ABB RAPID module: GM2694_96_A.mod

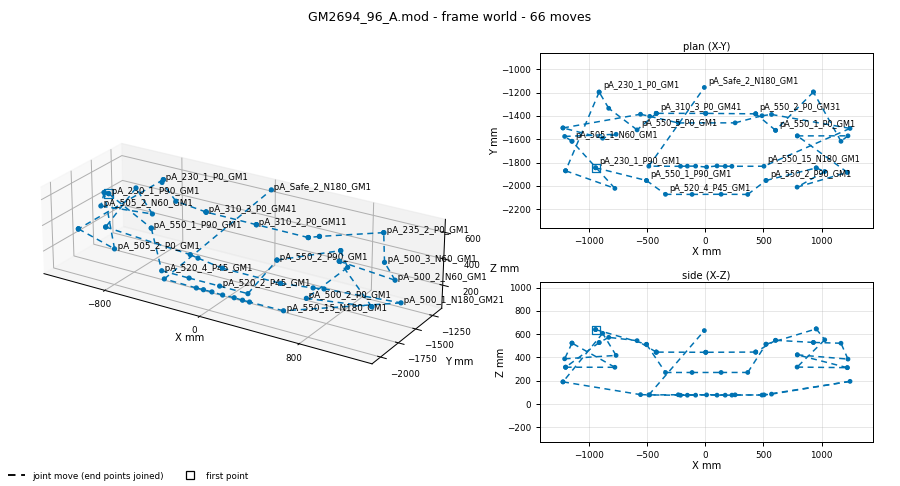
[picture p0: tool path of GM2694_96_A.mod in frame world, 66 of 72 moves have a stored position in this frame; points joined in program order, loops and branches not executed]
MODULE GM2694_96_A
	!Tool number
	TASK PERS wobjdata wobj_A_FD2:=[FALSE,TRUE,"STN2",[[0,0,0],[1,0,0,0]],[[-1.05287,-1136.44,433.383],[0.00113552,3.506E-06,-8.93971E-05,0.999999]]];

	!bailing room Jan 2013 Pad points
	CONST robtarget pTool_A_X1_FD2:=[[802.99,-1138.28,433.37],[1,2.43485E-05,-1.64211E-05,1.10567E-05],[-1,0,-1,1],[9E+09,9E+09,9E+09,9E+09,0.0243479,9E+09]];
	CONST robtarget pTool_A_X2_FD2:=[[-803.79,-1134.62,433.39],[1,2.20239E-05,-1.82688E-05,1.76728E-05],[-2,-1,0,1],[9E+09,9E+09,9E+09,9E+09,0.0253184,9E+09]];
	CONST robtarget pTool_A_Y1_FD2:=[[-3.61,-2246.56,433.25],[1,5.78314E-05,-1.3873E-05,6.83963E-06],[-2,-1,0,1],[9E+09,9E+09,9E+09,9E+09,0.0249386,9E+09]];

	TASK PERS wobjdata wobj_GM2694_96_A_GM2:=[FALSE,TRUE,"STN2",[[0,0,0],[1,0,0,0]],[[10.1671,-1103.71,380.343],[6.8405E-05,-0.000323021,-0.00059839,1]]];
	CONST robtarget GM2694_96_A_X1_GM2:=[[813.10,-1103.82,380.87],[1,4.78327E-05,-6.64294E-05,2.98321E-05],[-1,0,-1,1],[9E+09,9E+09,9E+09,9E+09,0.0311414,9E+09]];
	CONST robtarget GM2694_96_A_X2_GM2:=[[-790.92,-1103.60,379.83],[1,-3.83258E-05,0.000101328,3.79682E-05],[-2,-1,0,1],[9E+09,9E+09,9E+09,9E+09,0.0334623,9E+09]];
	CONST robtarget GM2694_96_A_Y1_GM2:=[[10.00,-2214.21,379.03],[1,0.000127688,0.000108138,1.82241E-05],[-1,0,-1,1],[9E+09,9E+09,9E+09,9E+09,0.00172991,9E+09]];

	!!TRUNNION AT P90
	CONST robtarget pA_230_1_P90_GM1:=[[950.40,741.13,260.17],[0.0696041,-3.9552E-05,8.47108E-05,-0.997575],[-2,-1,0,1],[9E+09,9E+09,9E+09,9E+09,89.9722,9E+09]];
	CONST robtarget pA_230_2_P90_GM1:=[[708.26,975.31,-115.95],[0.037863,-0.00102003,-0.000432508,-0.999282],[-2,-1,0,1],[9E+09,9E+09,9E+09,9E+09,44.9633,9E+09]];
	CONST robtarget pA_230_3_P90_GM1:=[[708.26,975.31,-115.95],[0.037863,-0.00102003,-0.000432508,-0.999282],[-2,-1,0,1],[9E+09,9E+09,9E+09,9E+09,44.9633,9E+09]];
	!
	CONST robtarget pA_235_1_P90_GM1:=[[-944.20,742.11,265.05],[0.0725762,0.000271763,-0.00166093,0.997362],[-1,0,-1,1],[9E+09,9E+09,9E+09,9E+09,89.9712,9E+09]];
	CONST robtarget pA_235_2_P90_GM1:=[[708.26,975.31,-115.95],[0.037863,-0.00102003,-0.000432508,-0.999282],[-2,-1,0,1],[9E+09,9E+09,9E+09,9E+09,44.9633,9E+09]];
	CONST robtarget pA_235_3_P90_GM1:=[[708.26,975.31,-115.95],[0.037863,-0.00102003,-0.000432508,-0.999282],[-2,-1,0,1],[9E+09,9E+09,9E+09,9E+09,44.9633,9E+09]];
	!
	CONST robtarget pA_310_1_P90_GM1:=[[353.14,746.45,293.52],[0.000120179,1.98777E-05,-0.0698146,0.99756],[-2,-1,0,1],[9E+09,9E+09,9E+09,9E+09,89.9669,9E+09]];
	CONST robtarget pA_310_2_P90_GM1:=[[120.58,746.64,293.48],[0.000119282,2.78364E-05,-0.0697897,0.997561],[-2,-1,0,1],[9E+09,9E+09,9E+09,9E+09,89.9659,9E+09]];
	CONST robtarget pA_310_3_P90_GM1:=[[-126.06,745.90,293.24],[8.89304E-05,2.54854E-06,-0.0697908,0.997561],[-1,0,-1,1],[9E+09,9E+09,9E+09,9E+09,89.9658,9E+09]];
	CONST robtarget pA_310_4_P90_GM1:=[[-355.40,745.70,293.41],[8.2894E-05,-9.32774E-06,-0.0697987,0.997561],[-1,0,-1,1],[9E+09,9E+09,9E+09,9E+09,89.9664,9E+09]];
	CONST robtarget pA_310_5_P90_GM1:=[[708.26,975.31,-115.95],[0.037863,-0.00102003,-0.000432508,-0.999282],[-2,-1,0,1],[9E+09,9E+09,9E+09,9E+09,44.9633,9E+09]];
	!
	CONST robtarget pA_550_1_P90_GM1:=[[513.56,850.46,133.60],[0.00698814,-3.27337E-05,8.28899E-05,-0.999976],[-2,-1,0,1],[9E+09,9E+09,9E+09,9E+09,89.9691,9E+09]];
	CONST robtarget pA_550_2_P90_GM1:=[[-512.81,849.94,133.81],[0.000446013,0.000442049,-0.000202557,-1],[-1,0,-1,1],[9E+09,9E+09,9E+09,9E+09,89.9679,9E+09]];
	CONST robtarget pA_550_3_P90_GM1:=[[335.13,751.81,293.47],[0.000114739,1.47188E-05,-0.069799,0.997561],[-2,-1,0,1],[9E+09,9E+09,9E+09,9E+09,89.9654,9E+09]];
	CONST robtarget pA_550_4_P90_GM1:=[[335.13,751.81,293.47],[0.000114739,1.47188E-05,-0.069799,0.997561],[-2,-1,0,1],[9E+09,9E+09,9E+09,9E+09,89.9654,9E+09]];
	CONST robtarget pA_550_5_P90_GM1:=[[335.13,751.81,293.47],[0.000114739,1.47188E-05,-0.069799,0.997561],[-2,-1,0,1],[9E+09,9E+09,9E+09,9E+09,89.9654,9E+09]];
	CONST robtarget pA_550_6_P90_GM1:=[[335.13,751.81,293.47],[0.000114739,1.47188E-05,-0.069799,0.997561],[-2,-1,0,1],[9E+09,9E+09,9E+09,9E+09,89.9654,9E+09]];
	CONST robtarget pA_550_7_P90_GM1:=[[335.13,751.81,293.47],[0.000114739,1.47188E-05,-0.069799,0.997561],[-2,-1,0,1],[9E+09,9E+09,9E+09,9E+09,89.9654,9E+09]];
	CONST robtarget pA_550_8_P90_GM1:=[[335.13,751.81,293.47],[0.000114739,1.47188E-05,-0.069799,0.997561],[-2,-1,0,1],[9E+09,9E+09,9E+09,9E+09,89.9654,9E+09]];
	CONST robtarget pA_550_9_P90_GM1:=[[335.13,751.81,293.47],[0.000114739,1.47188E-05,-0.069799,0.997561],[-2,-1,0,1],[9E+09,9E+09,9E+09,9E+09,89.9654,9E+09]];
	CONST robtarget pA_550_10_P90_GM1:=[[335.13,751.81,293.47],[0.000114739,1.47188E-05,-0.069799,0.997561],[-2,-1,0,1],[9E+09,9E+09,9E+09,9E+09,89.9654,9E+09]];

	!!TRUNNION AT P45
	CONST robtarget pA_520_1_P45_GM1:=[[-355.88,970.23,-108.48],[0.000696424,5.23204E-05,7.91609E-05,-1],[-1,0,-1,1],[9E+09,9E+09,9E+09,9E+09,60.0175,9E+09]];
	CONST robtarget pA_520_2_P45_GM1:=[[-127.19,968.94,-108.45],[0.000708875,4.20306E-05,8.75754E-05,-1],[-1,0,-1,1],[9E+09,9E+09,9E+09,9E+09,60.0162,9E+09]];
	CONST robtarget pA_520_3_P45_GM1:=[[122.35,969.96,-108.45],[0.000737368,8.10599E-05,7.36511E-05,-1],[-2,-1,0,1],[9E+09,9E+09,9E+09,9E+09,60.0186,9E+09]];
	CONST robtarget pA_520_4_P45_GM1:=[[350.43,969.49,-108.35],[0.000721682,5.88464E-05,9.34732E-05,-1],[-2,-1,0,1],[9E+09,9E+09,9E+09,9E+09,60.0185,9E+09]];
	CONST robtarget pA_520_5_P45_GM1:=[[921.24,100.58,148.76],[0.0161415,-0.451361,0.0125424,0.892107],[-2,-1,-1,1],[9E+09,9E+09,9E+09,9E+09,-0.0113089,9E+09]];
	CONST robtarget pA_520_6_P45_GM1:=[[921.24,100.58,148.76],[0.0161415,-0.451361,0.0125424,0.892107],[-2,-1,-1,1],[9E+09,9E+09,9E+09,9E+09,-0.0113089,9E+09]];
	CONST robtarget pA_520_7_P45_GM1:=[[921.24,100.58,148.76],[0.0161415,-0.451361,0.0125424,0.892107],[-2,-1,-1,1],[9E+09,9E+09,9E+09,9E+09,-0.0113089,9E+09]];
	CONST robtarget pA_520_8_P45_GM1:=[[921.24,100.58,148.76],[0.0161415,-0.451361,0.0125424,0.892107],[-2,-1,-1,1],[9E+09,9E+09,9E+09,9E+09,-0.0113089,9E+09]];

	!
	!!TRUNNION AT P0
	CONST robtarget pA_230_1_P0_GM1:=[[920.15,91.27,147.92],[0.00173565,-0.451157,0.0197843,0.892224],[-2,-1,-1,1],[9E+09,9E+09,9E+09,9E+09,-0.00898821,9E+09]];
	CONST robtarget pA_230_2_P0_GM1:=[[976.24,157.17,133.24],[0.366877,0.204171,0.141706,0.896457],[-2,0,-1,0],[9E+09,9E+09,9E+09,9E+09,-0.00983216,9E+09]];
	CONST robtarget pA_230_3_P0_GM1:=[[708.26,975.31,-115.95],[0.037863,-0.00102003,-0.000432508,-0.999282],[-2,-1,0,1],[9E+09,9E+09,9E+09,9E+09,44.9633,9E+09]];
	!
	CONST robtarget pA_235_1_P0_GM1:=[[-985.32,156.33,134.93],[0.353252,0.189241,-0.150106,-0.903809],[-1,-1,0,0],[9E+09,9E+09,9E+09,9E+09,-0.0140519,9E+09]];
	CONST robtarget pA_235_2_P0_GM1:=[[-919.56,90.31,147.84],[0.00214552,-0.450767,-0.018844,-0.89244],[-1,0,0,1],[9E+09,9E+09,9E+09,9E+09,-0.00962117,9E+09]];
	CONST robtarget pA_235_3_P0_GM1:=[[708.26,975.31,-115.95],[0.037863,-0.00102003,-0.000432508,-0.999282],[-2,-1,0,1],[9E+09,9E+09,9E+09,9E+09,44.9633,9E+09]];
	!
	CONST robtarget pA_310_1_P0_GM1:=[[-431.89,166.01,53.23],[0.000584676,-0.000297817,0.0434648,0.999055],[-1,0,-1,1],[9E+09,9E+09,9E+09,9E+09,-0.0200017,9E+09]];
	CONST robtarget pA_310_2_P0_GM1:=[[-7.04,167.31,54.58],[4.21115E-05,3.48116E-05,0.047325,0.99888],[-1,0,-1,1],[9E+09,9E+09,9E+09,9E+09,-0.0105073,9E+09]];
	CONST robtarget pA_310_3_P0_GM1:=[[430.45,166.27,53.78],[4.99449E-05,8.14198E-06,0.0448407,0.998994],[-2,-1,0,1],[9E+09,9E+09,9E+09,9E+09,-0.00962117,9E+09]];
	CONST robtarget pA_310_4_P0_GM1:=[[708.26,975.31,-115.95],[0.037863,-0.00102003,-0.000432508,-0.999282],[-2,-1,0,1],[9E+09,9E+09,9E+09,9E+09,44.9633,9E+09]];
	CONST robtarget pA_310_5_P0_GM1:=[[708.26,975.31,-115.95],[0.037863,-0.00102003,-0.000432508,-0.999282],[-2,-1,0,1],[9E+09,9E+09,9E+09,9E+09,44.9633,9E+09]];
	!
	CONST robtarget pA_500_1_P0_GM1:=[[-1210.79,780.16,-68.18],[0.00484054,0.124264,-0.0151395,0.992122],[-1,0,-1,1],[9E+09,9E+09,9E+09,9E+09,29.7818,9E+09]];
	CONST robtarget pA_500_2_P0_GM1:=[[-779.65,907.63,-62.79],[0.00917854,-0.069442,-0.0211429,0.99732],[-1,0,-1,1],[9E+09,9E+09,9E+09,9E+09,29.7802,9E+09]];
	CONST robtarget pA_500_3_P0_GM1:=[[708.26,975.31,-115.95],[0.037863,-0.00102003,-0.000432508,-0.999282],[-2,-1,0,1],[9E+09,9E+09,9E+09,9E+09,44.9633,9E+09]];
	CONST robtarget pA_500_4_P0_GM1:=[[708.26,975.31,-115.95],[0.037863,-0.00102003,-0.000432508,-0.999282],[-2,-1,0,1],[9E+09,9E+09,9E+09,9E+09,44.9633,9E+09]];
	CONST robtarget pA_500_5_P0_GM1:=[[708.26,975.31,-115.95],[0.037863,-0.00102003,-0.000432508,-0.999282],[-2,-1,0,1],[9E+09,9E+09,9E+09,9E+09,44.9633,9E+09]];
	!
	CONST robtarget pA_505_1_P0_GM1:=[[1208.02,767.29,-62.66],[0.00492163,-0.108695,0.00365501,0.994056],[-2,-1,0,1],[9E+09,9E+09,9E+09,9E+09,29.4206,9E+09]];
	CONST robtarget pA_505_2_P0_GM1:=[[785.04,918.35,-63.55],[0.0041262,0.0774671,-0.00566132,0.996971],[-2,-1,0,1],[9E+09,9E+09,9E+09,9E+09,29.4186,9E+09]];
	CONST robtarget pA_505_3_P0_GM1:=[[708.26,975.31,-115.95],[0.037863,-0.00102003,-0.000432508,-0.999282],[-2,-1,0,1],[9E+09,9E+09,9E+09,9E+09,44.9633,9E+09]];
	CONST robtarget pA_505_4_P0_GM1:=[[708.26,975.31,-115.95],[0.037863,-0.00102003,-0.000432508,-0.999282],[-2,-1,0,1],[9E+09,9E+09,9E+09,9E+09,44.9633,9E+09]];
	CONST robtarget pA_505_5_P0_GM1:=[[708.26,975.31,-115.95],[0.037863,-0.00102003,-0.000432508,-0.999282],[-2,-1,0,1],[9E+09,9E+09,9E+09,9E+09,44.9633,9E+09]];
	!
	CONST robtarget pA_520_1_P0_GM1:=[[708.26,975.31,-115.95],[0.037863,-0.00102003,-0.000432508,-0.999282],[-2,-1,0,1],[9E+09,9E+09,9E+09,9E+09,44.9633,9E+09]];
	CONST robtarget pA_520_2_P0_GM1:=[[708.26,975.31,-115.95],[0.037863,-0.00102003,-0.000432508,-0.999282],[-2,-1,0,1],[9E+09,9E+09,9E+09,9E+09,44.9633,9E+09]];
	CONST robtarget pA_520_3_P0_GM1:=[[708.26,975.31,-115.95],[0.037863,-0.00102003,-0.000432508,-0.999282],[-2,-1,0,1],[9E+09,9E+09,9E+09,9E+09,44.9633,9E+09]];
	CONST robtarget pA_520_4_P0_GM1:=[[708.26,975.31,-115.95],[0.037863,-0.00102003,-0.000432508,-0.999282],[-2,-1,0,1],[9E+09,9E+09,9E+09,9E+09,44.9633,9E+09]];
	CONST robtarget pA_520_5_P0_GM1:=[[708.26,975.31,-115.95],[0.037863,-0.00102003,-0.000432508,-0.999282],[-2,-1,0,1],[9E+09,9E+09,9E+09,9E+09,44.9633,9E+09]];
	!
	CONST robtarget pA_550_1_P0_GM1:=[[-594.77,419.41,166.72],[0.0335147,-0.547956,0.0209427,-0.835573],[-2,-1,0,1],[9E+09,9E+09,9E+09,9E+09,-0.0147692,9E+09]];
	CONST robtarget pA_550_2_P0_GM1:=[[-424.16,382.31,65.63],[3.20485E-06,-7.82063E-05,-2.24217E-05,1],[-1,0,-1,1],[9E+09,9E+09,9E+09,9E+09,-0.0182716,9E+09]];
	CONST robtarget pA_550_3_P0_GM1:=[[4.96,384.19,63.99],[1.51893E-05,-1.34389E-05,9.84778E-06,-1],[-1,0,-1,1],[9E+09,9E+09,9E+09,9E+09,-0.022618,9E+09]];
	CONST robtarget pA_550_4_P0_GM1:=[[429.59,384.16,65.78],[1.00484E-05,2.158E-05,-0.00545646,0.999985],[-2,-1,0,1],[9E+09,9E+09,9E+09,9E+09,-0.0183982,9E+09]];
	CONST robtarget pA_550_5_P0_GM1:=[[594.25,415.65,164.35],[0.0215819,-0.537366,-0.00959605,0.843019],[-1,0,-1,1],[9E+09,9E+09,9E+09,9E+09,-0.0207191,9E+09]];
	CONST robtarget pA_550_6_P0_GM1:=[[708.26,975.31,-115.95],[0.037863,-0.00102003,-0.000432508,-0.999282],[-2,-1,0,1],[9E+09,9E+09,9E+09,9E+09,44.9633,9E+09]];
	CONST robtarget pA_550_7_P0_GM1:=[[708.26,975.31,-115.95],[0.037863,-0.00102003,-0.000432508,-0.999282],[-2,-1,0,1],[9E+09,9E+09,9E+09,9E+09,44.9633,9E+09]];
	CONST robtarget pA_550_8_P0_GM1:=[[708.26,975.31,-115.95],[0.037863,-0.00102003,-0.000432508,-0.999282],[-2,-1,0,1],[9E+09,9E+09,9E+09,9E+09,44.9633,9E+09]];
	CONST robtarget pA_550_9_P0_GM1:=[[708.26,975.31,-115.95],[0.037863,-0.00102003,-0.000432508,-0.999282],[-2,-1,0,1],[9E+09,9E+09,9E+09,9E+09,44.9633,9E+09]];
	CONST robtarget pA_550_10_P0_GM1:=[[708.26,975.31,-115.95],[0.037863,-0.00102003,-0.000432508,-0.999282],[-2,-1,0,1],[9E+09,9E+09,9E+09,9E+09,44.9633,9E+09]];
	!
	!!TRUNNION AT N60
	CONST robtarget pA_500_1_N60_GM1:=[[-781.59,467.35,41.97],[0.00277233,0.0438581,0.00719055,-0.999008],[-1,0,-1,1],[9E+09,9E+09,9E+09,9E+09,-60.5108,9E+09]];
	CONST robtarget pA_500_2_N60_GM1:=[[-1216.32,466.78,4.87],[0.00374998,-0.10429,0.0069418,-0.994516],[-1,0,-1,1],[9E+09,9E+09,9E+09,9E+09,-60.5084,9E+09]];
	CONST robtarget pA_500_3_N60_GM1:=[[-1156.52,513.61,141.27],[0.004075,-0.00014402,1.15921E-05,-0.999992],[-1,0,-1,1],[9E+09,9E+09,9E+09,9E+09,-60.5074,9E+09]];
	CONST robtarget pA_500_4_N60_GM1:=[[708.26,975.31,-115.95],[0.037863,-0.00102003,-0.000432508,-0.999282],[-2,-1,0,1],[9E+09,9E+09,9E+09,9E+09,44.9633,9E+09]];
	CONST robtarget pA_500_5_N60_GM1:=[[708.26,975.31,-115.95],[0.037863,-0.00102003,-0.000432508,-0.999282],[-2,-1,0,1],[9E+09,9E+09,9E+09,9E+09,44.9633,9E+09]];
	!
	CONST robtarget pA_505_1_N60_GM1:=[[1153.28,513.79,143.87],[0.00515836,-2.20188E-05,1.67907E-05,-0.999987],[-2,-1,0,1],[9E+09,9E+09,9E+09,9E+09,-60.5039,9E+09]];
	CONST robtarget pA_505_2_N60_GM1:=[[1216.37,472.20,8.95],[0.00194678,0.139228,0.00768064,-0.990228],[-2,-1,0,1],[9E+09,9E+09,9E+09,9E+09,-60.506,9E+09]];
	CONST robtarget pA_505_3_N60_GM1:=[[774.68,453.62,38.06],[0.00982443,-0.0777471,0.000509252,-0.996924],[-2,-1,0,1],[9E+09,9E+09,9E+09,9E+09,-60.5055,9E+09]];
	CONST robtarget pA_505_4_N60_GM1:=[[708.26,975.31,-115.95],[0.037863,-0.00102003,-0.000432508,-0.999282],[-2,-1,0,1],[9E+09,9E+09,9E+09,9E+09,44.9633,9E+09]];
	CONST robtarget pA_505_5_N60_GM1:=[[708.26,975.31,-115.95],[0.037863,-0.00102003,-0.000432508,-0.999282],[-2,-1,0,1],[9E+09,9E+09,9E+09,9E+09,44.9633,9E+09]];
	!
	!!TRUNNION AT N180
	!
	CONST robtarget pA_310_1_N180_GM1:=[[-428.17,936.67,-352.11],[0.00042616,0.00356465,0.131785,0.991272],[-1,0,-1,1],[9E+09,9E+09,9E+09,9E+09,-171.335,9E+09]];
	CONST robtarget pA_310_2_N180_GM1:=[[-341.86,937.73,-374.62],[1.08478E-05,-1.53197E-05,6.13881E-05,-1],[-1,0,-1,1],[9E+09,9E+09,9E+09,9E+09,-171.333,9E+09]];
	CONST robtarget pA_310_3_N180_GM1:=[[-158.42,956.77,-359.65],[0.000398048,0.00352567,0.131823,0.991267],[-1,0,-1,1],[9E+09,9E+09,9E+09,9E+09,-171.335,9E+09]];
	CONST robtarget pA_310_4_N180_GM1:=[[-2.54,956.54,-360.66],[0.000394504,0.00351074,0.131803,0.99127],[-1,0,-1,1],[9E+09,9E+09,9E+09,9E+09,-171.335,9E+09]];
	CONST robtarget pA_310_5_N180_GM1:=[[158.74,956.26,-361.77],[0.000393889,0.00349563,0.131809,0.991269],[-2,-1,0,1],[9E+09,9E+09,9E+09,9E+09,-171.335,9E+09]];
	CONST robtarget pA_310_6_N180_GM1:=[[423.59,955.80,-363.58],[0.000400934,0.00347924,0.131815,0.991268],[-2,-1,0,1],[9E+09,9E+09,9E+09,9E+09,-171.335,9E+09]];
	CONST robtarget pA_310_7_N180_GM1:=[[492.88,939.60,-374.19],[4.56863E-05,-1.05492E-05,6.13342E-05,-1],[-2,-1,0,1],[9E+09,9E+09,9E+09,9E+09,-171.333,9E+09]];
	CONST robtarget pA_310_8_N180_GM1:=[[708.26,975.31,-115.95],[0.037863,-0.00102003,-0.000432508,-0.999282],[-2,-1,0,1],[9E+09,9E+09,9E+09,9E+09,44.9633,9E+09]];
	CONST robtarget pA_310_9_N180_GM1:=[[708.26,975.31,-115.95],[0.037863,-0.00102003,-0.000432508,-0.999282],[-2,-1,0,1],[9E+09,9E+09,9E+09,9E+09,44.9633,9E+09]];
	CONST robtarget pA_310_10_N180_GM1:=[[708.26,975.31,-115.95],[0.037863,-0.00102003,-0.000432508,-0.999282],[-2,-1,0,1],[9E+09,9E+09,9E+09,9E+09,44.9633,9E+09]];
	CONST robtarget pA_310_11_N180_GM1:=[[708.26,975.31,-115.95],[0.037863,-0.00102003,-0.000432508,-0.999282],[-2,-1,0,1],[9E+09,9E+09,9E+09,9E+09,44.9633,9E+09]];
	CONST robtarget pA_310_12_N180_GM1:=[[708.26,975.31,-115.95],[0.037863,-0.00102003,-0.000432508,-0.999282],[-2,-1,0,1],[9E+09,9E+09,9E+09,9E+09,44.9633,9E+09]];
	CONST robtarget pA_310_13_N180_GM1:=[[708.26,975.31,-115.95],[0.037863,-0.00102003,-0.000432508,-0.999282],[-2,-1,0,1],[9E+09,9E+09,9E+09,9E+09,44.9633,9E+09]];
	CONST robtarget pA_310_14_N180_GM1:=[[708.26,975.31,-115.95],[0.037863,-0.00102003,-0.000432508,-0.999282],[-2,-1,0,1],[9E+09,9E+09,9E+09,9E+09,44.9633,9E+09]];
	CONST robtarget pA_310_15_N180_GM1:=[[708.26,975.31,-115.95],[0.037863,-0.00102003,-0.000432508,-0.999282],[-2,-1,0,1],[9E+09,9E+09,9E+09,9E+09,44.9633,9E+09]];

	!
	CONST robtarget pA_500_1_N180_GM1:=[[-1243.50,381.67,-186.31],[0.706879,5.33573E-05,-2.34618E-06,-0.707334],[-1,-1,0,1],[9E+09,9E+09,9E+09,9E+09,-149.958,9E+09]];
	CONST robtarget pA_500_2_N180_GM1:=[[-1204.66,381.86,-186.15],[0.32853,-6.5977E-06,4.28364E-05,-0.944493],[-1,0,-1,1],[9E+09,9E+09,9E+09,9E+09,-149.952,9E+09]];
	CONST robtarget pA_500_3_N180_GM1:=[[-1137.07,519.96,141.43],[0.00405737,-1.80252E-05,5.82048E-05,-0.999991],[-1,0,-1,1],[9E+09,9E+09,9E+09,9E+09,-60.5062,9E+09]];
	CONST robtarget pA_500_4_N180_GM1:=[[708.26,975.31,-115.95],[0.037863,-0.00102003,-0.000432508,-0.999282],[-2,-1,0,1],[9E+09,9E+09,9E+09,9E+09,44.9633,9E+09]];
	CONST robtarget pA_500_5_N180_GM1:=[[708.26,975.31,-115.95],[0.037863,-0.00102003,-0.000432508,-0.999282],[-2,-1,0,1],[9E+09,9E+09,9E+09,9E+09,44.9633,9E+09]];
	!
	CONST robtarget pA_505_1_N180_GM1:=[[1247.14,383.93,-189.10],[0.701407,0.00116513,-0.000722366,0.71276],[-2,0,-1,1],[9E+09,9E+09,9E+09,9E+09,-149.95,9E+09]];
	CONST robtarget pA_505_2_N180_GM1:=[[1191.41,389.44,-184.88],[0.320474,-4.84084E-05,-0.000382623,0.947257],[-2,-1,0,1],[9E+09,9E+09,9E+09,9E+09,-149.948,9E+09]];
	CONST robtarget pA_505_3_N180_GM1:=[[775.04,447.88,42.59],[0.00201212,-0.0777562,-8.91676E-05,-0.99697],[-2,-1,0,1],[9E+09,9E+09,9E+09,9E+09,-60.5045,9E+09]];
	CONST robtarget pA_505_4_N180_GM1:=[[708.26,975.31,-115.95],[0.037863,-0.00102003,-0.000432508,-0.999282],[-2,-1,0,1],[9E+09,9E+09,9E+09,9E+09,44.9633,9E+09]];
	CONST robtarget pA_505_5_N180_GM1:=[[708.26,975.31,-115.95],[0.037863,-0.00102003,-0.000432508,-0.999282],[-2,-1,0,1],[9E+09,9E+09,9E+09,9E+09,44.9633,9E+09]];
	!
	CONST robtarget pA_550_1_N180_GM1:=[[-559.63,283.68,-295.55],[0.0147504,0.000861792,-0.0609037,-0.998034],[-1,0,-1,1],[9E+09,9E+09,9E+09,9E+09,-179.979,9E+09]];
	CONST robtarget pA_550_2_N180_GM1:=[[-478.05,294.69,-303.73],[0.0147591,0.000864438,-0.0609087,-0.998033],[-1,0,-1,1],[9E+09,9E+09,9E+09,9E+09,-179.979,9E+09]];
	CONST robtarget pA_550_3_N180_GM1:=[[-247.25,355.77,-301.46],[0.0147706,0.000817082,-0.060818,-0.998039],[-1,0,-1,1],[9E+09,9E+09,9E+09,9E+09,-179.973,9E+09]];
	CONST robtarget pA_550_4_N180_GM1:=[[240.75,356.48,-300.46],[0.0147869,0.000844929,-0.06086,-0.998036],[-2,-1,0,1],[9E+09,9E+09,9E+09,9E+09,-179.974,9E+09]];
	CONST robtarget pA_550_5_N180_GM1:=[[486.32,300.01,-301.48],[0.0147235,0.000873711,-0.06072,-0.998045],[-2,-1,0,1],[9E+09,9E+09,9E+09,9E+09,-179.984,9E+09]];
	CONST robtarget pA_550_6_N180_GM1:=[[564.91,282.00,-299.30],[0.0147448,0.000821824,-0.0615118,-0.997997],[-2,-1,0,1],[9E+09,9E+09,9E+09,9E+09,-179.973,9E+09]];
	CONST robtarget pA_550_7_N180_GM1:=[[493.76,727.96,-301.01],[0.0147461,-4.12593E-05,5.1514E-05,-0.999891],[-2,-1,0,1],[9E+09,9E+09,9E+09,9E+09,-179.974,9E+09]];
	CONST robtarget pA_550_8_N180_GM1:=[[221.63,728.95,-304.36],[0.000457518,-6.19018E-05,2.0639E-05,-1],[-2,-1,0,1],[9E+09,9E+09,9E+09,9E+09,-179.977,9E+09]];
	CONST robtarget pA_550_9_N180_GM1:=[[162.67,727.70,-303.88],[0.000453078,-2.12529E-05,3.2386E-06,-1],[-2,-1,0,1],[9E+09,9E+09,9E+09,9E+09,-179.974,9E+09]];
	CONST robtarget pA_550_10_N180_GM1:=[[92.00,727.46,-303.63],[0.452133,0.000350381,0.000126083,-0.891951],[-2,-1,0,1],[9E+09,9E+09,9E+09,9E+09,-179.978,9E+09]];
	CONST robtarget pA_550_11_N180_GM1:=[[-2.20,735.44,-301.12],[0.000517547,-2.66689E-05,1.49893E-05,-1],[-1,0,-1,1],[9E+09,9E+09,9E+09,9E+09,-179.978,9E+09]];
	CONST robtarget pA_550_12_N180_GM1:=[[-91.82,725.83,-303.61],[0.378753,-1.88066E-05,5.13943E-05,0.925498],[-1,0,-1,1],[9E+09,9E+09,9E+09,9E+09,-179.983,9E+09]];
	CONST robtarget pA_550_13_N180_GM1:=[[-161.93,728.67,-303.77],[0.000553349,1.03667E-05,1.92718E-05,-1],[-1,0,-1,1],[9E+09,9E+09,9E+09,9E+09,-179.982,9E+09]];
	CONST robtarget pA_550_14_N180_GM1:=[[-219.66,728.92,-303.46],[0.000559574,-1.19363E-05,1.4485E-05,-1],[-1,0,-1,1],[9E+09,9E+09,9E+09,9E+09,-179.98,9E+09]];
	CONST robtarget pA_550_15_N180_GM1:=[[-494.94,728.39,-301.20],[0.000540834,-3.59248E-05,3.30712E-05,-1],[-1,0,-1,1],[9E+09,9E+09,9E+09,9E+09,-179.983,9E+09]];
	CONST robtarget pA_550_16_N180_GM1:=[[335.13,751.81,293.47],[0.000114739,1.47188E-05,-0.069799,0.997561],[-2,-1,0,1],[9E+09,9E+09,9E+09,9E+09,89.9654,9E+09]];
	CONST robtarget pA_550_17_N180_GM1:=[[335.13,751.81,293.47],[0.000114739,1.47188E-05,-0.069799,0.997561],[-2,-1,0,1],[9E+09,9E+09,9E+09,9E+09,89.9654,9E+09]];
	CONST robtarget pA_550_18_N180_GM1:=[[335.13,751.81,293.47],[0.000114739,1.47188E-05,-0.069799,0.997561],[-2,-1,0,1],[9E+09,9E+09,9E+09,9E+09,89.9654,9E+09]];
	CONST robtarget pA_550_19_N180_GM1:=[[349.96,804.23,-301.33],[0.00200296,3.08902E-05,3.43427E-05,-0.999997],[-2,-1,0,1],[9E+09,9E+09,9E+09,9E+09,-179.995,9E+09]];
	CONST robtarget pA_550_20_N180_GM1:=[[122.28,635.67,-301.10],[0.000466004,-1.54693E-05,2.02502E-05,-1],[-2,-1,0,1],[9E+09,9E+09,9E+09,9E+09,-179.978,9E+09]];
	CONST robtarget pA_550_21_N180_GM1:=[[-128.60,758.45,-301.12],[0.000539466,-5.17921E-06,1.67757E-05,-0.999999],[-1,0,-1,1],[9E+09,9E+09,9E+09,9E+09,-179.978,9E+09]];
	CONST robtarget pA_550_22_N180_GM1:=[[-355.03,813.54,-301.49],[0.000634793,-1.21524E-05,2.88592E-06,-0.999999],[-1,0,-1,1],[9E+09,9E+09,9E+09,9E+09,-179.985,9E+09]];


    TASK PERS loaddata LoadGM2694_96A:=[950,[-60.2,-27.4,0],[1,0,0,0],0,0,111.4];


	CONST robtarget pA_Safe_1_P0_GM1:=[[74.00,88.93,243.71],[0.0279337,1.00884E-05,-5.36808E-05,0.999609],[-2,-1,0,1],[9E+09,9E+09,9E+09,9E+09,-0.012828,9E+09]];
	CONST robtarget pA_Safe_2_P0_GM1:=[[-1016.95,772.90,171.16],[0.0617771,0.0340987,-0.0116861,0.997439],[-1,0,-1,1],[9E+09,9E+09,9E+09,9E+09,46.4844,9E+09]];
	CONST robtarget pA_Safe_3_P0_GM1:=[[1206.65,483.09,309.68],[0.320571,-0.00610917,-0.0189757,0.947014],[-2,0,-1,1],[9E+09,9E+09,9E+09,9E+09,-0.012828,9E+09]];
	CONST robtarget pA_Safe_4_P0_GM1:=[[-867.31,489.74,258.29],[0.0101084,2.8178E-05,-5.44035E-05,0.999949],[-1,0,-1,1],[9E+09,9E+09,9E+09,9E+09,-0.012828,9E+09]];
	CONST robtarget pA_Safe_5_P0_GM1:=[[-867.31,489.74,258.29],[0.0101084,2.8178E-05,-5.44035E-05,0.999949],[-1,0,-1,1],[9E+09,9E+09,9E+09,9E+09,-0.012828,9E+09]];
	CONST robtarget pA_Safe_6_P0_GM1:=[[-867.31,489.74,258.29],[0.0101084,2.8178E-05,-5.44035E-05,0.999949],[-1,0,-1,1],[9E+09,9E+09,9E+09,9E+09,-0.012828,9E+09]];
	CONST robtarget pA_Safe_7_P0_GM1:=[[-867.31,489.74,258.29],[0.0101084,2.8178E-05,-5.44035E-05,0.999949],[-1,0,-1,1],[9E+09,9E+09,9E+09,9E+09,-0.012828,9E+09]];

	CONST robtarget pA_Safe_1_N180_GM1:=[[-1156.52,513.61,141.27],[0.00407409,-0.000144304,1.0892E-05,-0.999992],[-1,0,-1,1],[9E+09,9E+09,9E+09,9E+09,-60.5074,9E+09]];
	CONST robtarget pA_Safe_2_N180_GM1:=[[16.89,51.24,250.08],[0.00136107,-3.49227E-05,0.000388549,-0.999999],[-2,-1,0,1],[9E+09,9E+09,9E+09,9E+09,-149.948,9E+09]];
	CONST robtarget pA_Safe_3_N180_GM1:=[[16.88,51.24,250.08],[0.00136295,-3.96608E-05,0.000388216,-0.999999],[-2,-1,0,1],[9E+09,9E+09,9E+09,9E+09,33.5415,9E+09]];

	CONST robtarget pA_445_safe01_N180_FD2:=[[-1030.14,449.69,-57.42],[0.139634,-0.000906499,-0.000277604,-0.990202],[-1,0,-1,1],[9E+09,9E+09,9E+09,9E+09,-179.929,9E+09]];
	CONST robtarget pA_Safe_N90_2_FD2:=[[758.90,24.14,-68.10],[0.000305872,0.00120705,0.173796,0.98478],[-2,-1,0,1],[9E+09,9E+09,9E+09,9E+09,-58.1628,9E+09]];
	CONST robtarget pA_Safe_N90_3_FD2:=[[-894.81,518.59,346.96],[0.00406077,-2.99968E-05,5.05023E-05,-0.999991],[-1,0,-1,1],[9E+09,9E+09,9E+09,9E+09,-60.5068,9E+09]];

	 TASK PERS loaddata LoadCD4A:=[500,[-186.8,43.5,0],[1,0,0,0],0,0,111.6];
	 CONST robtarget pA_310_3_P0_GM11:=[[118.00,170.97,61.83],[1.50378E-05,9.39828E-05,0.349137,0.937071],[-2,-2,1,1],[9E+09,9E+09,9E+09,9E+09,-0.0116452,9E+09]];
	 CONST robtarget pA_310_3_P0_GM21:=[[-69.47,170.53,61.83],[0.000176017,0.000405876,-0.349724,-0.936852],[-1,-3,2,1],[9E+09,9E+09,9E+09,9E+09,-0.0116452,9E+09]];
	 CONST robtarget pA_310_3_P0_GM31:=[[418.63,150.23,76.65],[3.94592E-05,3.83899E-05,-0.0695289,0.99758],[-2,-1,0,1],[9E+09,9E+09,9E+09,9E+09,-0.0114764,9E+09]];
	 CONST robtarget pA_Safe_1_P0_GM11:=[[-133.98,370.35,115.62],[1.43539E-06,-0.000153872,0.000326658,-1],[-1,0,-1,1],[9E+09,9E+09,9E+09,9E+09,-0.0260345,9E+09]];
	 CONST robtarget pA_Safe_1_P0_GM21:=[[87.56,371.82,110.31],[7.20878E-05,-3.64463E-05,-9.16335E-05,-1],[-2,-1,0,1],[9E+09,9E+09,9E+09,9E+09,-0.024642,9E+09]];
	 CONST robtarget pA_550_2_P0_GM11:=[[-211.67,381.61,65.74],[1.42713E-05,-3.53997E-05,-2.62415E-05,1],[-1,0,-1,1],[9E+09,9E+09,9E+09,9E+09,-0.0221101,9E+09]];
	 CONST robtarget pA_Safe_1_P0_GM31:=[[164.45,382.29,65.86],[6.94651E-05,-4.51965E-05,0.00013405,-1],[-2,-1,0,1],[9E+09,9E+09,9E+09,9E+09,-0.0139238,9E+09]];
	 CONST robtarget pA_Safe_1_P0_GM41:=[[289.52,382.81,66.11],[0.000101662,4.79564E-06,0.000242721,-1],[-2,-1,0,1],[9E+09,9E+09,9E+09,9E+09,-0.0150632,9E+09]];
	 CONST robtarget pA_550_2_P0_GM21:=[[-305.63,381.18,65.79],[5.51581E-05,-2.16418E-05,9.71512E-05,-1],[-1,0,-1,1],[9E+09,9E+09,9E+09,9E+09,-0.0158227,9E+09]];
	 CONST robtarget pA_550_3_P0_GM11:=[[-500.29,821.09,60.62],[4.47715E-05,-0.000119148,3.95027E-05,-1],[-1,0,-1,1],[9E+09,9E+09,9E+09,9E+09,-0.0229133,9E+09]];
	 CONST robtarget pA_550_3_P0_GM21:=[[544.17,820.66,59.57],[0.00895683,0.000798268,0.0896038,0.995937],[-2,-1,0,1],[9E+09,9E+09,9E+09,9E+09,-0.0271753,9E+09]];
	 CONST robtarget pA_550_3_P0_GM31:=[[-305.89,827.79,64.06],[2.70716E-05,0.000193981,-6.75608E-05,1],[-1,0,-1,1],[9E+09,9E+09,9E+09,9E+09,-0.0257828,9E+09]];
	 CONST robtarget pA_550_3_P0_GM41:=[[302.59,831.97,64.05],[1.58097E-05,0.000186113,-7.45256E-05,0.999999],[-2,-1,0,1],[9E+09,9E+09,9E+09,9E+09,-0.0270909,9E+09]];
	 CONST robtarget pA_550_3_P0_GM51:=[[-5.14,829.43,64.07],[2.59921E-06,0.000183846,-7.04278E-05,1],[-1,0,-1,1],[9E+09,9E+09,9E+09,9E+09,-0.0283975,9E+09]];
	 CONST robtarget pA_Safe_1_P0_GM51:=[[-127.64,383.92,64.03],[6.11971E-06,-3.47988E-05,4.01987E-05,-1],[-1,0,-1,1],[9E+09,9E+09,9E+09,9E+09,-0.0240934,9E+09]];
	 CONST robtarget pA_550_3_P0_GM61:=[[130.08,384.50,64.02],[1.053E-05,-2.85946E-05,3.58546E-05,-1],[-2,-1,0,1],[9E+09,9E+09,9E+09,9E+09,-0.02422,9E+09]];

	 CONST robtarget GM2694_96_Gusset_01_SP:=[[-815,859.64,93.81],[0.0013179,-0.00552133,0.00178163,-0.999982],[1,0,-1,1],[9E+09,9E+09,9E+09,9E+09,0.015823,9E+09]];
     CONST robtarget GM2694_96_Gusset_02_SP:=[[281.25,861.95,82.15],[0.00129516,-0.00551131,0.00180622,-0.999982],[0,-1,0,1],[9E+09,9E+09,9E+09,9E+09,0.0157386,9E+09]];
     CONST robtarget GM2694_96_Gusset_01_WD:=[[-811.48,890.57,93.87],[0.00131668,-0.00553775,0.00177641,-0.999982],[1,0,-1,1],[9E+09,9E+09,9E+09,9E+09,0.0151493,9E+09]];
     CONST robtarget GM2694_96_Gusset_02_WD:=[[273.52,893.74,82.36],[0.00129268,-0.00549839,0.00180798,-0.999982],[0,-1,0,1],[9E+09,9E+09,9E+09,9E+09,0.0154025,9E+09]];
     CONST robtarget pA_550_3_P0_GM71:=[[-545.52,818.66,63.48],[0.00897472,0.000804225,0.0896081,0.995937],[-1,0,-1,1],[9E+09,9E+09,9E+09,9E+09,-0.0267955,9E+09]];
     CONST robtarget pA_310_1_N180_GM11:=[[-338.19,957.13,-358.33],[0.000418656,0.0035354,0.131795,0.991271],[-1,0,-1,1],[9E+09,9E+09,9E+09,9E+09,-171.335,9E+09]];
     CONST robtarget pA_310_3_N180_GM11:=[[-158.42,956.77,-359.64],[0.000397421,0.00352659,0.131822,0.991267],[-1,0,-1,1],[9E+09,9E+09,9E+09,9E+09,-171.335,9E+09]];
     CONST robtarget pA_310_1_N180_GM21:=[[465.80,946.56,-361.39],[0.000402916,0.0034825,0.131821,0.991268],[-2,-1,0,1],[9E+09,9E+09,9E+09,9E+09,-171.335,9E+09]];
     CONST robtarget pA_500_1_N180_GM11:=[[890.09,487.13,227.80],[0.0204307,0.000339386,0.000584551,-0.999791],[-2,-1,0,1],[9E+09,9E+09,9E+09,9E+09,-92.6919,9E+09]];
     CONST robtarget pA_550_2_P0_GM31:=[[-424.16,278.02,65.62],[8.3166E-06,-7.73541E-05,-1.88321E-05,1],[-1,0,-1,1],[9E+09,9E+09,9E+09,9E+09,-0.0178075,9E+09]];
     CONST robtarget pA_310_1_P0_GM11:=[[-424.17,278.01,65.61],[1.22766E-05,-6.86796E-05,-1.4273E-05,1],[-1,0,-1,1],[9E+09,9E+09,9E+09,9E+09,-0.0170057,9E+09]];
     CONST robtarget pA_550_3_P0_GM81:=[[4.96,274,64.04],[2.6719E-05,2.86862E-06,2.83524E-05,-1],[-1,0,-1,1],[9E+09,9E+09,9E+09,9E+09,-0.0218162,9E+09]];
     CONST robtarget pA_310_2_P0_GM11:=[[4.97,274,64.02],[2.5033E-05,3.47895E-06,2.26458E-05,-1],[-1,0,-1,1],[9E+09,9E+09,9E+09,9E+09,-0.0211832,9E+09]];
     CONST robtarget pA_550_4_P0_GM11:=[[429.58,274,65.78],[1.04349E-05,2.35173E-05,-0.00545569,0.999985],[-2,-1,0,1],[9E+09,9E+09,9E+09,9E+09,-0.0179762,9E+09]];
     CONST robtarget pA_310_3_P0_GM41:=[[429.56,273.97,65.73],[5.88644E-06,-1.57577E-05,0.00543819,-0.999985],[-2,-1,0,1],[9E+09,9E+09,9E+09,9E+09,-0.0173855,9E+09]];
     CONST robtarget pA_505_1_N180_GM11:=[[1231.00,399.56,-189.02],[0.390023,0.000811047,-0.00107786,0.920805],[-2,0,-1,1],[9E+09,9E+09,9E+09,9E+09,-149.951,9E+09]];
     CONST robtarget pA_500_1_N180_GM21:=[[-1233.96,403.31,-186.24],[0.386385,8.59202E-05,4.33185E-05,-0.922338],[-1,-1,0,1],[9E+09,9E+09,9E+09,9E+09,-149.958,9E+09]];
	!

	PROC rGM2694_96_A_Welding()
			SetGO TaskActive, 1;
            rSpeed_Override;
			!ClkReset clock_A_Weld_cycle;
			!ClkStart clock_A_Weld_cycle;
			!
			!PulseDO OpenCellAInnerDoor;

			ActUnit STN2;
			!DeactUnit STN1;
			MechUnitLoad Stn2, 1, LoadGM2694_96A;
			WaitDI CellAInnerDoorOpened ,1;
			!
			ClkReset clock_A_Weld_cycle;
			ClkStart clock_A_Weld_cycle;

		IF RobotProduction = 1 THEN
			vProduction := [7500,7500,7500,180];
			vHome := [2500, 2500, 2500, 90];
	  	ELSE
			vProduction := [200,100,100,20];
			vHome := [100, 100, 100, 10];
	  	ENDIF
			!
			rMoveToCell_A;
			Set PFOAirJet;
			!
			MoveAbsJ pA_Load\NoEOffs, vProduction, z200, t3D_PFO\WObj:=wobj0;
			PulseDO WeldStarted;
			Set LaserRequest;
			IF TAClampsSafePFO = 0 Stop;
			!
			AccSet 100,100;

			MoveJ pA_230_1_P90_GM1,vProduction,fine,t3D_PFO\WObj:=wobj_GM2694_96_A_GM2;
			!WaitTime 0.5;
			IF AS520_PP = 1 Then
			!
			!K2
			SetGO PFOProgReq, 712;
			SetGO LaserProgReq, 61;
			MoveJ pA_230_1_P90_GM1,vProduction,fine,t3D_PFO\WObj:=wobj_GM2694_96_A_GM2;
			rPFO_Dimpling;

			ENDIF

			MoveJ pA_550_1_P90_GM1,vProduction,fine,t3D_PFO\WObj:=wobj_GM2694_96_A_GM2;

            IF AW550PP = 1 Then
			!K2
			SetGO PFOProgReq, 510;
			SetGO LaserProgReq, 61;
			MoveJ pA_550_1_P90_GM1,vProduction,fine,t3D_PFO\WObj:=wobj_GM2694_96_A_GM2;
		    rPFO_Welding;

            ENDIF



            !AW510


            IF GM2696_A_Selected = 1 AND GM2694_A_Selected = 0 AND   AW500PP = 1 Then

			SetGO LaserProgReq, 128;
			MoveJ pA_520_4_P45_GM1, vProduction, fine, t3D_PFO\WObj:=wobj_GM2694_96_A_GM2;
			rPFO_Welding;

            SetGO LaserProgReq, 128;
			MoveJ pA_520_3_P45_GM1, vProduction, fine, t3D_PFO\WObj:=wobj_GM2694_96_A_GM2;
			rPFO_Welding;

			SetGO LaserProgReq, 128;
			MoveJ pA_520_2_P45_GM1, vProduction, fine, t3D_PFO\WObj:=wobj_GM2694_96_A_GM2;
			rPFO_Welding;

            SetGO LaserProgReq, 128;
			MoveJ pA_520_1_P45_GM1, vProduction, fine, t3D_PFO\WObj:=wobj_GM2694_96_A_GM2;
			rPFO_Welding;

            ENDIF


            !
			MoveJ pA_550_2_P90_GM1,vProduction,fine,t3D_PFO\WObj:=wobj_GM2694_96_A_GM2;
			IF AW550PP = 1 Then
			!
			!M2
			SetGO PFOProgReq, 516;
			SetGO LaserProgReq, 61;
			MoveJ pA_550_2_P90_GM1,vProduction,fine,t3D_PFO\WObj:=wobj_GM2694_96_A_GM2;
			rPFO_Welding;

			ENDIF

			MoveJ pA_235_1_P90_GM1,vProduction,fine,t3D_PFO\WObj:=wobj_GM2694_96_A_GM2;

			IF AS525_2PP = 1 Then
			!
			!M2
			SetGO PFOProgReq, 718;
			SetGO LaserProgReq, 61;
			MoveJ pA_235_1_P90_GM1,vProduction,fine,t3D_PFO\WObj:=wobj_GM2694_96_A_GM2;
			rPFO_Dimpling;

			ENDIF

			!MoveJ pA_Safe_2_P0_GM1, vProduction, z200, t3D_PFO\WObj:=wobj_GM2694_96_A_GM2;
			MoveJ pA_Safe_2_P0_GM1, vProduction, z200, t3D_PFO\WObj:=wobj_GM2694_96_A_GM2;



            IF AW545PP = 1 THEN

			!H5
			SetGO PFOProgReq, 499;
			SetGO LaserProgReq, 61;
			MoveJ pA_500_2_P0_GM1,vProduction,fine,t3D_PFO\WObj:=wobj_GM2694_96_A_GM2;
			rPFO_Welding;

			ENDIF
			!
			IF AW545PP = 1 AND GM2696_A_Selected = 0 AND GM2694_A_Selected = 1 THEN

			!G1   G2-1   G2-2
			SetGO LaserProgReq, 66;
			MoveJ pA_500_1_P0_GM1,vProduction,fine,t3D_PFO\WObj:=wobj_GM2694_96_A_GM2;
			rPFO_Welding;

            ENDIF
			!
			IF AW545PP = 1 AND GM2696_A_Selected = 1 AND GM2694_A_Selected = 0 THEN

			!G1   G2-1   G2-2
			SetGO LaserProgReq, 129;
			MoveJ pA_500_1_P0_GM1,vProduction,fine,t3D_PFO\WObj:=wobj_GM2694_96_A_GM2;
			rPFO_Welding;

			ENDIF


            MoveJ pA_500_1_N60_GM1,vProduction,fine,t3D_PFO\WObj:=wobj_GM2694_96_A_GM2;

			IF AW545PP = 1 Then
			!
			!H6
			SetGO PFOProgReq, 500;
			SetGO LaserProgReq, 61;
			MoveJ pA_500_1_N60_GM1,vProduction,fine,t3D_PFO\WObj:=wobj_GM2694_96_A_GM2;
			rPFO_Welding;
			!
			!G3
			SetGO PFOProgReq, 492;
			SetGO LaserProgReq, 61;
			MoveJ pA_500_2_N60_GM1,vProduction,fine,t3D_PFO\WObj:=wobj_GM2694_96_A_GM2;
			rPFO_Welding;
			!
			!F4
			SetGO LaserProgReq, 111;
			MoveJ pA_500_3_N60_GM1,vProduction,fine,t3D_PFO\WObj:=wobj_GM2694_96_A_GM2;
			rPFO_Welding;

			ENDIF


			IF AS525_2PP = 1 Then


			!F4
			SetGO PFOProgReq, 686;
			SetGO LaserProgReq, 61;
			MoveJ pA_235_2_P0_GM1,vProduction,fine,t3D_PFO\WObj:=wobj_GM2694_96_A_GM2;
			rPFO_Dimpling;

			ENDIF


			MoveJ pA_235_2_P0_GM1,vProduction,fine,t3D_PFO\WObj:=wobj_GM2694_96_A_GM2;
			!AW550
			MoveJ pA_550_1_P0_GM1,vProduction,fine,t3D_PFO\WObj:=wobj_GM2694_96_A_GM2;
			IF AW550PP = 1 Then

			SetGO LaserProgReq, 106;
			MoveJ pA_550_1_P0_GM1,vProduction,fine,t3D_PFO\WObj:=wobj_GM2694_96_A_GM2;
			rPFO_Welding;

			SetGO PFOProgReq, 515;
			SetGO LaserProgReq, 61;
			!MoveJ pA_550_2_P0_GM1,vProduction,fine,t3D_PFO\WObj:=wobj_GM2694_96_A_GM2;
			MoveJ pA_550_2_P0_GM31, vPRODUCTION, fine, t3D_PFO\WObj:=wobj_GM2694_96_A_GM2;
			rPFO_Welding;

			ENDIF

			!AS500
			!MoveJ pA_310_1_P0_GM1,vProduction,fine,t3D_PFO\WObj:=wobj_GM2694_96_A_GM2;
			MoveJ pA_310_1_P0_GM11, vPRODUCTION, fine, t3D_PFO\WObj:=wobj_GM2694_96_A_GM2;

			IF AS500PP = 1 Then

			!M1
			SetGO PFOProgReq, 717;
			SetGO LaserProgReq, 61;
			WaitTime 0.1;
			!MoveJ pA_310_1_P0_GM1,vProduction,fine,t3D_PFO\WObj:=wobj_GM2694_96_A_GM2;
			MoveJ pA_310_1_P0_GM11, vPRODUCTION, fine, t3D_PFO\WObj:=wobj_GM2694_96_A_GM2;
			rPFO_Welding;

			!J1
			SetGO PFOProgReq, 703;
			SetGO LaserProgReq, 61;
			!MoveJ pA_310_2_P0_GM1,vProduction,fine,t3D_PFO\WObj:=wobj_GM2694_96_A_GM2;
			MoveJ pA_310_2_P0_GM11, vPRODUCTION, fine, t3D_PFO\WObj:=wobj_GM2694_96_A_GM2;
			rPFO_Welding;

			ENDIF

			!AW550
			!MoveJ pA_550_3_P0_GM1, vProduction, fine, t3D_PFO\WObj:=wobj_GM2694_96_A_GM2;
			MoveJ pA_550_3_P0_GM81, vPRODUCTION, fine, t3D_PFO\WObj:=wobj_GM2694_96_A_GM2;

			IF AW550PP = 1 Then

			!J1
			SetGO LaserProgReq, 107;
			!MoveJ pA_550_3_P0_GM1, vProduction, fine, t3D_PFO\WObj:=wobj_GM2694_96_A_GM2;
			WaitTime 0.1;
			MoveJ pA_550_3_P0_GM81, vPRODUCTION, fine, t3D_PFO\WObj:=wobj_GM2694_96_A_GM2;
			rPFO_Welding;

			ENDIF

			!AS500
			!MoveJ pA_310_3_P0_GM1,vProduction,fine,t3D_PFO\WObj:=wobj_GM2694_96_A_GM2;
			MoveJ pA_310_3_P0_GM41, vPRODUCTION, fine, t3D_PFO\WObj:=wobj_GM2694_96_A_GM2;

			IF AS500PP = 1 Then
			!
			!K1
			SetGO PFOProgReq, 711;
			SetGO LaserProgReq, 61;
			!MoveJ pA_310_3_P0_GM1,vProduction,fine,t3D_PFO\WObj:=wobj_GM2694_96_A_GM2;
			MoveJ pA_310_3_P0_GM41, vPRODUCTION, fine, t3D_PFO\WObj:=wobj_GM2694_96_A_GM2;
			rPFO_Dimpling;

			ENDIF

			!AW550
			!MoveJ pA_550_4_P0_GM1,vProduction,fine,t3D_PFO\WObj:=wobj_GM2694_96_A_GM2;
			MoveJ pA_550_4_P0_GM11, vPRODUCTION, fine, t3D_PFO\WObj:=wobj_GM2694_96_A_GM2;

			IF AW550PP = 1 Then

			!K1
			SetGO PFOProgReq, 509;
			SetGO LaserProgReq, 61;
			WaitTime 0.1;
			!MoveJ pA_550_4_P0_GM1,vProduction,fine,t3D_PFO\WObj:=wobj_GM2694_96_A_GM2;
			MoveJ pA_550_4_P0_GM11, vPRODUCTION, fine, t3D_PFO\WObj:=wobj_GM2694_96_A_GM2;
			rPFO_Welding;

			SetGO LaserProgReq, 108;
			MoveJ pA_550_5_P0_GM1,vProduction,fine,t3D_PFO\WObj:=wobj_GM2694_96_A_GM2;
			rPFO_Welding;

			ENDIF

			!AS520
			MoveJ [[838.00,230.44,192.72],[0.0040269,-0.473827,-0.0060738,0.880588],[-2,-1,-1,1],[9E+09,9E+09,9E+09,9E+09,-0.011731,9E+09]], vPRODUCTION, z200, t3D_PFO\WObj:=wobj_GM2694_96_A_GM2;
			MoveJ pA_230_1_P0_GM1,vProduction,fine,t3D_PFO\WObj:=wobj_GM2694_96_A_GM2;

			IF AS520_PP = 1 Then
			!C4
			!MoveJ [[838.00,230.44,192.72],[0.0040269,-0.473827,-0.0060738,0.880588],[-2,-1,-1,1],[9E+09,9E+09,9E+09,9E+09,-0.011731,9E+09]], vPRODUCTION, z200, t3D_PFO\WObj:=wobj_GM2694_96_A_GM2;
			SetGO PFOProgReq, 668;
			SetGO LaserProgReq, 140;
			MoveJ pA_230_1_P0_GM1,vProduction,fine,t3D_PFO\WObj:=wobj_GM2694_96_A_GM2;
			rPFO_Dimpling;

			!SetGO PFOProgReq, 716;
			!SetGO LaserProgReq, 140;
			!MoveJ pA_230_2_P0_GM1,vProduction,fine,t3D_PFO\WObj:=wobj_GM2694_96_A_GM2;
			!rPFO_Dimpling;
			!
			ENDIF

			!MoveJ pA_230_2_P0_GM1,vProduction,fine,t3D_PFO\WObj:=wobj_GM2694_96_A_GM2;

			MoveJ pA_505_1_P0_GM1,vProduction,fine,t3D_PFO\WObj:=wobj_GM2694_96_A_GM2;

			IF AW540PP = 1 AND GM2696_A_Selected = 0 AND GM2694_A_Selected = 1 Then

			!D1   D2-1    D2-2
			SetGO LaserProgReq, 67;
			MoveJ pA_505_1_P0_GM1,vProduction,fine,t3D_PFO\WObj:=wobj_GM2694_96_A_GM2;
			rPFO_Welding;

            ENDIF

            IF AW540PP = 1 AND GM2696_A_Selected = 1 AND GM2694_A_Selected = 0 Then

			!D1   D2-1    D2-2
			SetGO LaserProgReq, 132;
			MoveJ pA_505_1_P0_GM1,vProduction,fine,t3D_PFO\WObj:=wobj_GM2694_96_A_GM2;
			rPFO_Welding;

            ENDIF

            IF AW540PP = 1 THEN

			!E5
			SetGO PFOProgReq, 479;
			SetGO LaserProgReq, 61;
			MoveJ pA_505_2_P0_GM1,vProduction,fine,t3D_PFO\WObj:=wobj_GM2694_96_A_GM2;
			rPFO_Welding;

			ENDIF

			MoveJ pA_505_1_N60_GM1,vProduction,fine,t3D_PFO\WObj:=wobj_GM2694_96_A_GM2;
			IF AW540PP = 1 Then

			SetGO LaserProgReq, 109;
			MoveJ pA_505_1_N60_GM1,vProduction,fine,t3D_PFO\WObj:=wobj_GM2694_96_A_GM2;
			rPFO_Welding;

			SetGO PFOProgReq, 472;
			SetGO LaserProgReq, 61;
			MoveJ pA_505_2_N60_GM1,vProduction,fine,t3D_PFO\WObj:=wobj_GM2694_96_A_GM2;
			rPFO_Welding;
			!E6
			SetGO PFOProgReq, 480;
			SetGO LaserProgReq, 61;
			MoveJ pA_505_3_N60_GM1,vProduction,fine,t3D_PFO\WObj:=wobj_GM2694_96_A_GM2;
			rPFO_Welding;
			!
			ENDIF

			!MoveJ pA_Safe_1_N180_GM1, vProduction, z50, t3D_PFO\WObj:=wobj_GM2694_96_A_GM2;
			!MoveJ pA_500_1_N180_GM1,vProduction,fine,t3D_PFO\WObj:=wobj_GM2694_96_A_GM2;

		    MoveJ pA_500_1_N180_GM11, vPRODUCTION, z200, t3D_PFO\WObj:=wobj_GM2694_96_A_GM2;


            !MoveJ pA_505_1_N180_GM1,vProduction,fine,t3D_PFO\WObj:=wobj_GM2694_96_A_GM2;
            MoveJ pA_505_1_N180_GM11, vPRODUCTION, fine, t3D_PFO\WObj:=wobj_GM2694_96_A_GM2;

            IF AW540PP = 1 Then
			!
			SetGO LaserProgReq, 75;
			!MoveJ pA_505_1_N180_GM1,vProduction,fine,t3D_PFO\WObj:=wobj_GM2694_96_A_GM2;
			MoveJ pA_505_1_N180_GM11, vPRODUCTION, fine, t3D_PFO\WObj:=wobj_GM2694_96_A_GM2;
			rPFO_Welding;
			!
			ENDIF


			! AW550

			IF AW550PP = 1 Then

			SetGO LaserProgReq, 115;
			MoveJ pA_550_6_N180_GM1,vProduction,fine,t3D_PFO\WObj:=wobj_GM2694_96_A_GM2;
			rPFO_Welding;

            SetGO PFOProgReq, 473;
			SetGO LaserProgReq, 61;
			MoveJ pA_550_5_N180_GM1,vProduction,fine,t3D_PFO\WObj:=wobj_GM2694_96_A_GM2;
			rPFO_Welding;

            SetGO LaserProgReq, 114;
			MoveJ pA_550_4_N180_GM1,vProduction,fine,t3D_PFO\WObj:=wobj_GM2694_96_A_GM2;
			rPFO_Welding;

			SetGO LaserProgReq, 113;
			MoveJ pA_550_3_N180_GM1,vProduction,fine,t3D_PFO\WObj:=wobj_GM2694_96_A_GM2;
			rPFO_Welding;

			SetGO PFOProgReq, 493;
			SetGO LaserProgReq, 61;
			MoveJ pA_550_2_N180_GM1,vProduction,fine,t3D_PFO\WObj:=wobj_GM2694_96_A_GM2;
			rPFO_Welding;

            SetGO LaserProgReq, 112;
			MoveJ pA_550_1_N180_GM1,vProduction,fine,t3D_PFO\WObj:=wobj_GM2694_96_A_GM2;
			rPFO_Welding;

            ENDIF


        IF AW545PP = 1 Then
			!
			SetGO LaserProgReq, 68;
			!MoveJ pA_500_1_N180_GM1,vProduction,fine,t3D_PFO\WObj:=wobj_GM2694_96_A_GM2;
			MoveJ pA_500_1_N180_GM21, vPRODUCTION, fine, t3D_PFO\WObj:=wobj_GM2694_96_A_GM2;
			rPFO_Welding;
			!
			ENDIF

          IF AW550PP = 1 Then

            SetGO PFOProgReq, 483;
			SetGO LaserProgReq, 61;
			MoveJ pA_550_15_N180_GM1,vProduction,fine,t3D_PFO\WObj:=wobj_GM2694_96_A_GM2;
			rPFO_Welding;

            SetGO PFOProgReq, 401;
			SetGO LaserProgReq, 61;
			MoveJ pA_550_14_N180_GM1,vProduction,fine,t3D_PFO\WObj:=wobj_GM2694_96_A_GM2;
			rPFO_Welding;

			SetGO PFOProgReq, 404;
			SetGO LaserProgReq, 61;
			MoveJ pA_550_13_N180_GM1,vProduction,fine,t3D_PFO\WObj:=wobj_GM2694_96_A_GM2;
			rPFO_Welding;

            SetGO LaserProgReq, 70;
			MoveJ pA_550_12_N180_GM1,vProduction,fine,t3D_PFO\WObj:=wobj_GM2694_96_A_GM2;
			rPFO_Welding;

            SetGO LaserProgReq, 116;
			MoveJ pA_550_11_N180_GM1,vProduction,fine,t3D_PFO\WObj:=wobj_GM2694_96_A_GM2;
			rPFO_Welding;

            SetGO LaserProgReq, 69;
			MoveJ pA_550_10_N180_GM1,vProduction,fine,t3D_PFO\WObj:=wobj_GM2694_96_A_GM2;
			rPFO_Welding;

			SetGO PFOProgReq, 425;
			SetGO LaserProgReq, 61;
			MoveJ pA_550_9_N180_GM1,vProduction,fine,t3D_PFO\WObj:=wobj_GM2694_96_A_GM2;
			rPFO_Welding;

            SetGO PFOProgReq, 428;
			SetGO LaserProgReq, 61;
			MoveJ pA_550_8_N180_GM1,vProduction,fine,t3D_PFO\WObj:=wobj_GM2694_96_A_GM2;
			rPFO_Welding;

			SetGO PFOProgReq, 463;
			SetGO LaserProgReq, 61;
			MoveJ pA_550_7_N180_GM1,vProduction,fine,t3D_PFO\WObj:=wobj_GM2694_96_A_GM2;
			rPFO_Welding;

			ENDIF


			MoveJ pA_Safe_2_N180_GM1, vProduction, z200, t3D_PFO\WObj:=wobj_GM2694_96_A_GM2;

			Reset PFOAirJet;
			Reset LaserRequest;
			AccSet 100,100;

			MoveAbsJ pA_Safe_N107\NoEOffs, vProduction, z200, t3D_PFO\WObj:=wobj0;
			MoveAbsJ pA_Safe_N069\NoEOffs, vProduction, z200, t3D_PFO\WObj:=wobj0;
			PulseDO\PLength:=1, WeldCompleted;
			MoveAbsJ pA_Safe_N031\NoEOffs, vProduction, z200, t3D_PFO\WObj:=wobj0;
			MoveAbsJ pA_Safe_P007\NoEOffs, vProduction, z200, t3D_PFO\WObj:=wobj0;
			MoveAbsJ pA_Unload\NoEOffs, vProduction, Fine, t3D_PFO\WObj:=wobj0;
			PulseDO\PLength:= 1.0, ToolAatLoadingPos;
         IF ToolAChangeReq = 1 THEN
                 rTool_A_Change_Pos;
         ENDIF
			DeactUnit STN2;
			!WaitTime 0.25;
			!!
			!
			ClkStop clock_A_Weld_cycle;
			TPWrite "A Welding Cycle Time (ms) = " \Num:= ClkRead(clock_A_Weld_cycle)*1000;
			nA_Weld_Cycle_Time:= ClkRead(clock_A_Weld_cycle)*1000;
			SetGO TaskActive, 0;
	ENDPROC
ENDMODULE
